(* IEC 61131-3 sources: strictdoc/tests/integration/features/source_code_traceability/_file_types/65_st_structured_text, 1 file *)

(* ---- file.st ---- *)
FUNCTION_BLOCK FB_Test
VAR_INPUT
	i_xA: BOOL;
	i_xB: BOOL;
END_VAR
VAR_OUTPUT
	o_xX: BOO;
END_VAR

// --- BEGIN IMPLEMENTATION ---
// @relation(REQ-001, scope=range_start)
IF i_xA AND i_xB THEN
	o_xX := TRUE;
ELSE
	o_xX := FALSE;
END_IF
// @relation(REQ-001, scope=range_end)
